// TIA Portal project "Quantum" (V16)

(* hardware
DEVICE "S7-1200 station_1"  S7-1200 Station
   slot 0: "Rack_0"  S7-1200 Rack  Rack  V1.0
   slot 1: "Quantum_Deshidratador"  CPU 1214C DC/DC/DC  6ES7 214-1AG40-0XB0  V4.4
   slot 101: "CM 1241 (RS422/485)_1"  6ES7 241-1CH32-0XB0  V2.1
*)

// ===== PLC "Quantum_Deshidratador"  CPU 1214C DC/DC/DC =====
// protected blocks, not shown: "MODULO_SECADOR"

VAR_GLOBAL   // PLC tag table "Default tag table"
   "Iniciar_Manual" AT %I0.0 : Bool;
   "Detener_Manual" AT %I0.1 : Bool;
   "Raw_Temperatura" AT %IW64 : Int;
   "Raw_Humedad" AT %IW66 : Int;
   "Deshidratador" AT %Q0.0 : Bool;
   "Actuador_Matte" AT %Q0.4 : Bool;
   "Ventiladores" AT %Q0.1 : Bool;
   "Resistencias" AT %Q0.5 : Bool;
   "Sensor_Modbus" AT %Q0.3 : Bool;
   "Sensor_HT" AT %Q0.2 : Bool;
   "System_Byte" AT %MB1 : Byte;
   "FirstScan" AT %M1.0 : Bool;
   "DiagStatusUpdate" AT %M1.1 : Bool;
   "AlwaysTRUE" AT %M1.2 : Bool;
   "AlwaysFALSE" AT %M1.3 : Bool;
   "Clock_Byte" AT %MB0 : Byte;
   "Clock_10Hz" AT %M0.0 : Bool;
   "Clock_5Hz" AT %M0.1 : Bool;
   "Clock_2.5Hz" AT %M0.2 : Bool;
   "Clock_2Hz" AT %M0.3 : Bool;
   "Clock_1.25Hz" AT %M0.4 : Bool;
   "Clock_1Hz" AT %M0.5 : Bool;
   "Clock_0.625Hz" AT %M0.6 : Bool;
   "Clock_0.5Hz" AT %M0.7 : Bool;
   "Control_Byte" AT %MB2 : Byte;
   "Detener" AT %M2.0 : Bool;
   "Iniciar" AT %M2.1 : Bool;
   "Pausar" AT %M2.2 : Bool;
   "Activar_Deshidratador" AT %M2.3 : Bool;
   "Limite_Matte" AT %M2.6 : Bool;
   "Sensor_Modbus_Manual" AT %M2.4 : Bool;
   "Set_Point_Deshidratador" AT %MD4 : Real;
   "Set_Point_Humedad" AT %MD8 : Real;
   "Iniciar_Pulse" AT %M40.0 : Bool;
   "Detener_Pulse" AT %M40.1 : Bool;
   "Guardar_Datos" AT %M40.2 : Bool;
   "Data_Log_Write_Error" AT %M40.3 : Bool;
   "Data_Log_Write_Busy" AT %M40.4 : Bool;
   "Data_Log_Write_Done" AT %M40.5 : Bool;
   "Data_Log_Write_Status" AT %MW96 : Word;
   "Clock_0.016Hz" AT %M40.6 : Bool;
   "Ret_Val" AT %MW98 : Int;
   "Sensor_HT_Manual" AT %M2.5 : Bool;
   "Actuador_Manual" AT %M2.7 : Bool;
   "Activar_Actuador" AT %M3.0 : Bool;
   "Tag_1" AT %M41.1 : Bool;
   "Habilitar_Matte" AT %M3.1 : Bool;
   "Set_Point_Limite" AT %MD12 : Real;
   "Humedad_Material_D11" AT %MD100 : Real;
   "Humedad_Material_D13" AT %MD104 : Real;
   "Humedad_Material_D16" AT %MD108 : Real;
   "Temp_D13" AT %MD114 : Real;
   "Temp_Matte" AT %MD118 : Real;
   "Hum_Matte" AT %MD62 : Real;
   "Temp_D11" AT %MD112 : Real;
   "Temp_Matte_Aux" AT %MD66 : Real;
   "Clock_Matte_Manual" AT %M41.2 : Bool;
   "Humedad_Material_D11_Ajuste" AT %MD70 : Real;
   "Humedad_Material_D13_Ajuste" AT %MD74 : Real;
   "Humedad_Material_D16_Ajuste" AT %MD78 : Real;
   "Hum_Matte_Aux" AT %MD82 : Real;
   "Random_Real_Seconds" AT %MD86 : Real;
   "Random_Status" AT %MW90 : Int;
   "Random_Sub_Status" AT %MW92 : Int;
   "Random_Error" AT %M3.2 : Bool;
   "Clock_Pulse" AT %M3.3 : Bool;
   "Randon_Dint_Seconds" AT %MD94 : DInt;
   "Tiempo_Histeresis_D1" AT %MD14 : Time;
   "Set_Point_Deshidratador1_Inicial" AT %MD18 : Real;
   "Set_Point_Deshidratador1_Intermedia" AT %MD22 : Real;
   "Set_Point_Deshidratador1_Final" AT %MD24 : Real;
   "Set_Point_Humedad_D1_Inicial" AT %MD28 : Real;
   "Set_Point_Humedad_D1_Intermedia" AT %MD32 : Real;
   "Set_Point_Humedad_D1_Final" AT %MD36 : Real;
   "Detener_Desde_Modo_Preset" AT %M41.3 : Bool;
   "Detener_Desde_Modo_Temporidado" AT %M41.4 : Bool;
END_VAR

VAR_GLOBAL CONSTANT   // PLC tag table "Default tag table"
   "Set_Point_Temp_Default" : Real := 55.0;
   "Set_Pont_Hum_Default" : Real := 5.0;
   "Set_Point_Lim_Default" : Real := -16.0;
   "Aux_Hum_D1" : Real := 10.0;
   "Aux_Hum_D4" : Real := 25.0;
   "Aux_Hum_D8" : Real := 25.0;
END_VAR

DATA_BLOCK "Modos_Operacion"   // DB32
{ S7_Optimized_Access := 'TRUE' }
VERSION : 0.1
   VAR RETAIN
      Modo_Preset_D1 : Bool := true;
      Momento_Actual_D1 : Int;
   END_VAR
BEGIN
END_DATA_BLOCK

DATA_BLOCK "Alarmas"   // DB44
{ S7_Optimized_Access := 'FALSE' }
VERSION : 0.1
   VAR
      Alarma_Fin_Operacion : Bool;
      Alarma_Fallo_Deh : Bool;
   END_VAR
BEGIN
END_DATA_BLOCK

// folder: Data Logging

DATA_BLOCK "CREAR_DB"   // DB7
{ S7_Optimized_Access := 'TRUE' }
VERSION : 0.1
   VAR
      records : UDInt := 17280;
      "name" : String := 'logging';
      id : DWord := 1;
      headers : String := 'HumD11,HumD13,HumD16,TempD11,TempD13,HumMatte,TempMatte';
      data : Struct
         humD11 : Real;
         humD13 : Real;
         humD16 : Real;
         tempD11 : Real;
         tempD13 : Real;
         humMatte : Real;
         tempMatte : Real;
      END_STRUCT;
      done : Bool;
      busy : Bool := true;
      error : Bool;
      status : Word;
   END_VAR
BEGIN
END_DATA_BLOCK

DATA_BLOCK "DATOS_VARIABLES"   // DB8
{ S7_Optimized_Access := 'FALSE' }
VERSION : 0.1
   VAR
      humD11 : Real;
      humD13 : Real;
      humD16 : Real;
      tempD11 : Real;
      tempD13 : Real;
      humMatte : Real;
      tempMatte : Real;
      dehRunning : Bool;
   END_VAR
BEGIN
END_DATA_BLOCK

DATA_BLOCK "Control_Log_DB"   // DB33
{ S7_Optimized_Access := 'FALSE' }
VERSION : 0.1
   VAR
      Iniciar_Log : Bool;
      Almacenar_Logs : Bool;
      Teminar_Log : Bool;
   END_VAR
BEGIN
END_DATA_BLOCK

// folder: Matte

DATA_BLOCK "DATOS_MODSEC"   // DB13
{ S7_Optimized_Access := 'TRUE' }
VERSION : 0.1
   VAR
      SimuHR : Int;
   END_VAR
   VAR RETAIN
      "Paso Control HR" : Time := T#5000ms;
      "Paso Grafica" : Time := T#10ms;
      "CRECIMIENTO HR" : Real := 80.0;
      TempMinHR : Real := 22.0;
   END_VAR
   VAR
      TempInf : Real := 0.0;
      TempSup : Real := 100.0;
      TempFilt : Real;
      TempFiltJP : Real;
      HRAux : Real;
      HRAuxJP : Real;
      HRFilt : Real;
      HRSim : Int;
      TempSim : Int;
      ProporcionHumedad : Real := 0.9;
      TempFiltCuar : Real;
      HRFiltCuar : Real;
      HRAuxCuar : Real;
   END_VAR
BEGIN
END_DATA_BLOCK

// folder: Modbus

DATA_BLOCK "MB_CONFIG"   // DB9
{ S7_Optimized_Access := 'FALSE' }
VERSION : 0.1
   VAR
      Again : Bool;
      Req : Bool;
      Mb_Addr : UInt := 1;
      Mode : USInt := 0;
      Data_Addr : UDInt := 40001;
      Data_Len : UInt := 5;
      Done : Bool;
      Busy : Bool;
      Error : Bool;
      Status : Word;
      Error_Status : Word;
      "Step" : Int := 1;
   END_VAR
BEGIN
END_DATA_BLOCK

DATA_BLOCK "MB_DATA_BUFFER"   // DB10
{ S7_Optimized_Access := 'FALSE' }
VERSION : 0.1
   VAR
      REGISTERS : Array[0..4] of UInt;
   END_VAR
BEGIN
END_DATA_BLOCK

DATA_BLOCK "MB_LOAD"   // DB11
{ S7_Optimized_Access := 'FALSE' }
VERSION : 0.1
   VAR
      Baud : UDInt := 9600;
      Parity : UDInt;
      Done : Bool;
      Error : Bool;
      Status : Word;
      Done_Stored : Bool;
      Error_Stored : Bool;
      Status_Error : Word;
   END_VAR
BEGIN
END_DATA_BLOCK

// folder: Sensores

DATA_BLOCK "Escalado_Temp_DB"   // DB18
{ S7_Optimized_Access := 'TRUE' }
VERSION : 0.1
// stored: InstanceOfName Escalado_Temp
"Escalado_Temp"
BEGIN
END_DATA_BLOCK

DATA_BLOCK "Conversor_4-20_0-20_DB"   // DB19
{ S7_Optimized_Access := 'TRUE' }
VERSION : 0.1
// stored: InstanceOfName Conversor_4-20_0-20
"Conversor_4-20_0-20"
BEGIN
END_DATA_BLOCK

DATA_BLOCK "Sensor_HR_DB"   // DB20
{ S7_Optimized_Access := 'TRUE' }
VERSION : 0.1
// stored: InstanceOfName Sensor_HR
"Sensor_HR"
BEGIN
END_DATA_BLOCK

DATA_BLOCK "Filtro_Promedio_DB"   // DB21
{ S7_Optimized_Access := 'TRUE' }
VERSION : 0.1
// stored: InstanceOfName Filtro_Promedio
"Filtro_Promedio"
BEGIN
END_DATA_BLOCK

DATA_BLOCK "Conversor_4-20_0-20_DB_1"   // DB22
{ S7_Optimized_Access := 'TRUE' }
VERSION : 0.1
// stored: InstanceOfName Conversor_4-20_0-20
"Conversor_4-20_0-20"
BEGIN
END_DATA_BLOCK

DATA_BLOCK "Simulacion_HR_DB"   // DB23
{ S7_Optimized_Access := 'TRUE' }
VERSION : 0.1
// stored: InstanceOfName Simulacion_HR
"Simulacion_HR"
BEGIN
END_DATA_BLOCK

DATA_BLOCK "Prom_FilterV2_DB"   // DB25
{ S7_Optimized_Access := 'TRUE' }
VERSION : 0.1
// stored: InstanceOfName Prom_FilterV2
"Prom_FilterV2"
BEGIN
END_DATA_BLOCK

DATA_BLOCK "Calibracion_Sensores"   // DB31
{ S7_Optimized_Access := 'TRUE' }
VERSION : 0.1
   VAR
      Ajuste_D11 : Real := 1.0;
      Ajuste_D13 : Real := 1.0;
      Ajuste_D16 : Real := 1.0;
      Ajuste_T1 : Real := 1.0;
   END_VAR
BEGIN
END_DATA_BLOCK

// folder: System blocks/Program resources

DATA_BLOCK "Paso_DB"   // DB1
{ S7_Optimized_Access := 'TRUE' }
AUTHOR : Simatic
FAMILY : IEC
NAME : IEC_TMR
VERSION : 1.0
// stored: InstanceOfName IEC_TIMER
"IEC_TIMER"
BEGIN
END_DATA_BLOCK

DATA_BLOCK "IEC_Timer_0_DB"   // DB14
{ S7_Optimized_Access := 'TRUE' }
AUTHOR : Simatic
FAMILY : IEC
NAME : IEC_TMR
VERSION : 1.0
// stored: InstanceOfName IEC_TIMER
"IEC_TIMER"
BEGIN
END_DATA_BLOCK

DATA_BLOCK "IEC_Timer_0_DB_1"   // DB16
{ S7_Optimized_Access := 'TRUE' }
AUTHOR : Simatic
FAMILY : IEC
NAME : IEC_TMR
VERSION : 1.0
// stored: InstanceOfName IEC_TIMER
"IEC_TIMER"
BEGIN
END_DATA_BLOCK

DATA_BLOCK "IEC_Timer_0_DB_2"   // DB17
{ S7_Optimized_Access := 'TRUE' }
AUTHOR : Simatic
FAMILY : IEC
NAME : IEC_TMR
VERSION : 1.0
// stored: InstanceOfName IEC_TIMER
"IEC_TIMER"
BEGIN
END_DATA_BLOCK

DATA_BLOCK "Timer_SimHR_DB"   // DB24
{ S7_Optimized_Access := 'TRUE' }
AUTHOR : Simatic
FAMILY : IEC
NAME : IEC_TMR
VERSION : 1.0
// stored: InstanceOfName IEC_TIMER
"IEC_TIMER"
BEGIN
END_DATA_BLOCK

DATA_BLOCK "IEC_Timer_0_DB_3"   // DB26
{ S7_Optimized_Access := 'TRUE' }
AUTHOR : Simatic
FAMILY : IEC
NAME : IEC_TMR
VERSION : 1.0
// stored: InstanceOfName IEC_TIMER
"IEC_TIMER"
BEGIN
END_DATA_BLOCK

DATA_BLOCK "Control_Temporizado"   // DB27
{ S7_Optimized_Access := 'TRUE' }
AUTHOR : Simatic
FAMILY : IEC
NAME : IEC_TMR
VERSION : 1.0
// stored: InstanceOfName IEC_TIMER
"IEC_TIMER"
BEGIN
END_DATA_BLOCK

DATA_BLOCK "IEC_Timer_0_DB_5"   // DB28
{ S7_Optimized_Access := 'TRUE' }
AUTHOR : Simatic
FAMILY : IEC
NAME : IEC_TMR
VERSION : 1.0
// stored: InstanceOfName IEC_TIMER
"IEC_TIMER"
BEGIN
END_DATA_BLOCK

DATA_BLOCK "IEC_Timer_0_DB_6"   // DB29
{ S7_Optimized_Access := 'TRUE' }
AUTHOR : Simatic
FAMILY : IEC
NAME : IEC_TMR
VERSION : 1.0
// stored: InstanceOfName IEC_TIMER
"IEC_TIMER"
BEGIN
END_DATA_BLOCK

DATA_BLOCK "IEC_Timer_0_DB_7"   // DB30
{ S7_Optimized_Access := 'TRUE' }
AUTHOR : Simatic
FAMILY : IEC
NAME : IEC_TMR
VERSION : 1.0
// stored: InstanceOfName IEC_TIMER
"IEC_TIMER"
BEGIN
END_DATA_BLOCK

DATA_BLOCK "Histeresis_Timer"   // DB34
{ S7_Optimized_Access := 'TRUE' }
AUTHOR : Simatic
FAMILY : IEC
NAME : IEC_TMR
VERSION : 1.0
// stored: InstanceOfName IEC_TIMER
"IEC_TIMER"
BEGIN
END_DATA_BLOCK

// folder: (top level)

FUNCTION "Control_Maestro" : Void   // FC1, SCL
{ S7_Optimized_Access := 'TRUE' }
VERSION : 0.1
   VAR_INPUT
      Temperatura : Int;
      SetValue : Int;
   END_VAR
   VAR_OUTPUT
      HabilitarControl : Bool;
      Resitencias : Bool;
   END_VAR
   VAR CONSTANT
      Hysteresis : Int := 1;
   END_VAR
BEGIN
   IF #Temperatura < #SetValue AND NOT #HabilitarControl OR #Temperatura > #SetValue + #Hysteresis AND #HabilitarControl THEN
       #HabilitarControl := FALSE;
       #Resitencias := TRUE;
   ELSE
       #HabilitarControl := TRUE;
       #Resitencias := FALSE;
   END_IF;
END_FUNCTION

ORGANIZATION_BLOCK "Main"   // OB1, LAD, ProgramCycle
TITLE = "Main Program Sweep (Cycle)"
{ S7_Optimized_Access := 'TRUE' }
VERSION : 0.1
   VAR_INPUT
      Initial_Call : Bool;   // Initial call of this OB
      Remanence : Bool;   // =True, if remanent data are available
   END_VAR
   VAR_TEMP   // added for the SCL form of the ladder/FBD networks
      _w1 : Bool;
      _w2 : Bool;
      _w3 : Bool;
   END_VAR
BEGIN

REGION Network 1: Iniciar Detener
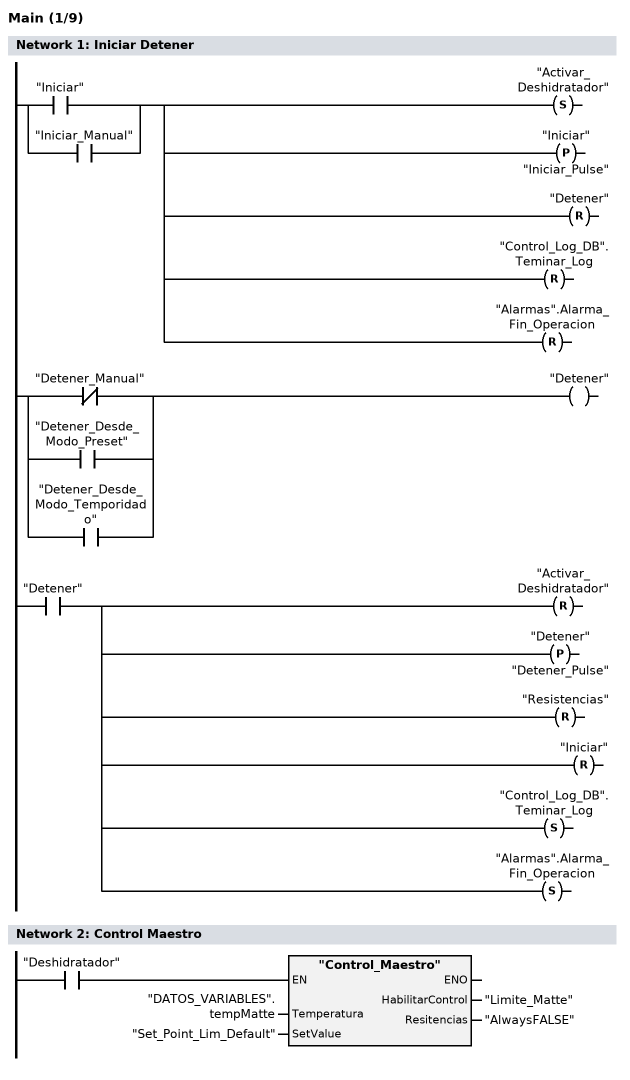
   #_w1 := "Iniciar" OR "Iniciar_Manual";
   IF #_w1 THEN "Activar_Deshidratador" := TRUE; END_IF;
   "Iniciar" := #_w1 AND NOT "Iniciar_Pulse";   // rising edge
   "Iniciar_Pulse" := #_w1;
   IF #_w1 THEN
       "Detener" := FALSE;
       "Control_Log_DB".Teminar_Log := FALSE;
       "Alarmas".Alarma_Fin_Operacion := FALSE;
   END_IF;
   "Detener" := NOT "Detener_Manual" OR "Detener_Desde_Modo_Preset" OR "Detener_Desde_Modo_Temporidado";
   IF "Detener" THEN "Activar_Deshidratador" := FALSE; END_IF;
   #_w2 := "Detener";
   #_w3 := "Detener";
   "Detener" := #_w2 AND NOT "Detener_Pulse";   // rising edge
   "Detener_Pulse" := #_w2;
   IF #_w3 THEN
       "Resistencias" := FALSE;
       "Iniciar" := FALSE;
       "Control_Log_DB".Teminar_Log := TRUE;
       "Alarmas".Alarma_Fin_Operacion := TRUE;
   END_IF;
END_REGION

REGION Network 2: Control Maestro
   RUNG wire#powerrail
      Contact( "Deshidratador" )
      "Control_Maestro"(Temperatura := "DATOS_VARIABLES".tempMatte, SetValue := "Set_Point_Lim_Default", HabilitarControl => "Limite_Matte", Resitencias => "AlwaysFALSE")
   END_RUNG
   // the same network as SCL:
   IF "Deshidratador" THEN
       "Control_Maestro"(Temperatura := "DATOS_VARIABLES".tempMatte,
                         SetValue := "Set_Point_Lim_Default",
                         HabilitarControl => "Limite_Matte",
                         Resitencias => "AlwaysFALSE");
   END_IF;
END_REGION

REGION Network 3: Matte
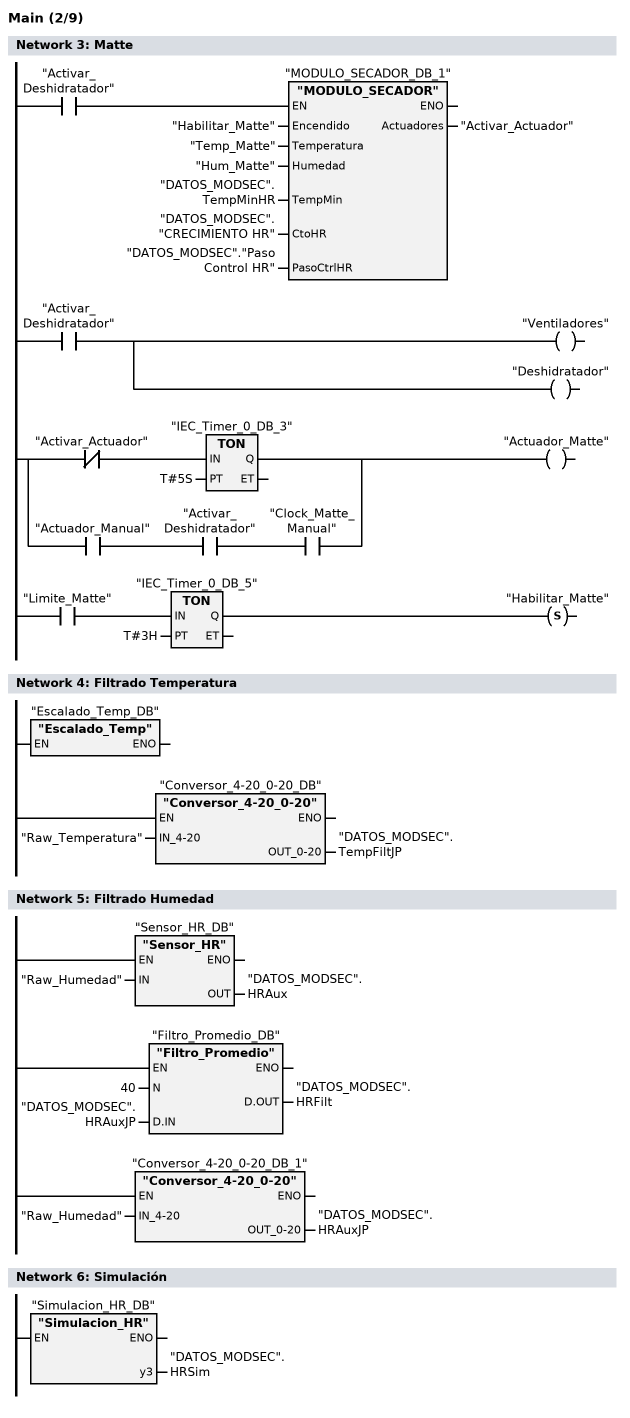
   IF "Activar_Deshidratador" THEN
       "MODULO_SECADOR_DB_1"(Encendido := "Habilitar_Matte",   // "MODULO_SECADOR"
                             Temperatura := "Temp_Matte",
                             Humedad := "Hum_Matte",
                             TempMin := "DATOS_MODSEC".TempMinHR,
                             CtoHR := "DATOS_MODSEC"."CRECIMIENTO HR",
                             PasoCtrlHR := "DATOS_MODSEC"."Paso Control HR",
                             Actuadores => "Activar_Actuador");
   END_IF;
   "Ventiladores" := "Activar_Deshidratador";
   "Deshidratador" := "Activar_Deshidratador";
   "IEC_Timer_0_DB_3".TON(IN := NOT "Activar_Actuador", PT := T#5S);
   "Actuador_Matte" := "IEC_Timer_0_DB_3".Q OR ("Actuador_Manual" AND "Activar_Deshidratador" AND "Clock_Matte_Manual");
   "IEC_Timer_0_DB_5".TON(IN := "Limite_Matte", PT := T#3H);
   IF "IEC_Timer_0_DB_5".Q THEN "Habilitar_Matte" := TRUE; END_IF;
END_REGION

REGION Network 4: Filtrado Temperatura
   RUNG wire#powerrail
      "Escalado_Temp_DB"()
   END_RUNG
   RUNG wire#powerrail
      "Conversor_4-20_0-20_DB"("IN_4-20" := "Raw_Temperatura", "OUT_0-20" => "DATOS_MODSEC".TempFiltJP)
   END_RUNG
   // the same network as SCL:
   "Escalado_Temp_DB"();   // "Escalado_Temp"
   "Conversor_4-20_0-20_DB"("IN_4-20" := "Raw_Temperatura", "OUT_0-20" => "DATOS_MODSEC".TempFiltJP);   // "Conversor_4-20_0-20"
END_REGION

REGION Network 5: Filtrado Humedad
   RUNG wire#powerrail
      "Sensor_HR_DB"(IN := "Raw_Humedad", OUT => "DATOS_MODSEC".HRAux)
   END_RUNG
   RUNG wire#powerrail
      "Filtro_Promedio_DB"(N := 40, "D.IN" := "DATOS_MODSEC".HRAuxJP, "D.OUT" => "DATOS_MODSEC".HRFilt)
   END_RUNG
   RUNG wire#powerrail
      "Conversor_4-20_0-20_DB_1"("IN_4-20" := "Raw_Humedad", "OUT_0-20" => "DATOS_MODSEC".HRAuxJP)
   END_RUNG
   // the same network as SCL:
   "Sensor_HR_DB"(IN := "Raw_Humedad", OUT => "DATOS_MODSEC".HRAux);   // "Sensor_HR"
   "Filtro_Promedio_DB"(N := 40, "D.IN" := "DATOS_MODSEC".HRAuxJP, "D.OUT" => "DATOS_MODSEC".HRFilt);   // "Filtro_Promedio"
   "Conversor_4-20_0-20_DB_1"("IN_4-20" := "Raw_Humedad", "OUT_0-20" => "DATOS_MODSEC".HRAuxJP);   // "Conversor_4-20_0-20"
END_REGION

REGION Network 6: Simulación
   RUNG wire#powerrail
      "Simulacion_HR_DB"(y3 => "DATOS_MODSEC".HRSim)
   END_RUNG
   // the same network as SCL:
   "Simulacion_HR_DB"(y3 => "DATOS_MODSEC".HRSim);   // "Simulacion_HR"
END_REGION

REGION Network 7: Manejo Sensorica
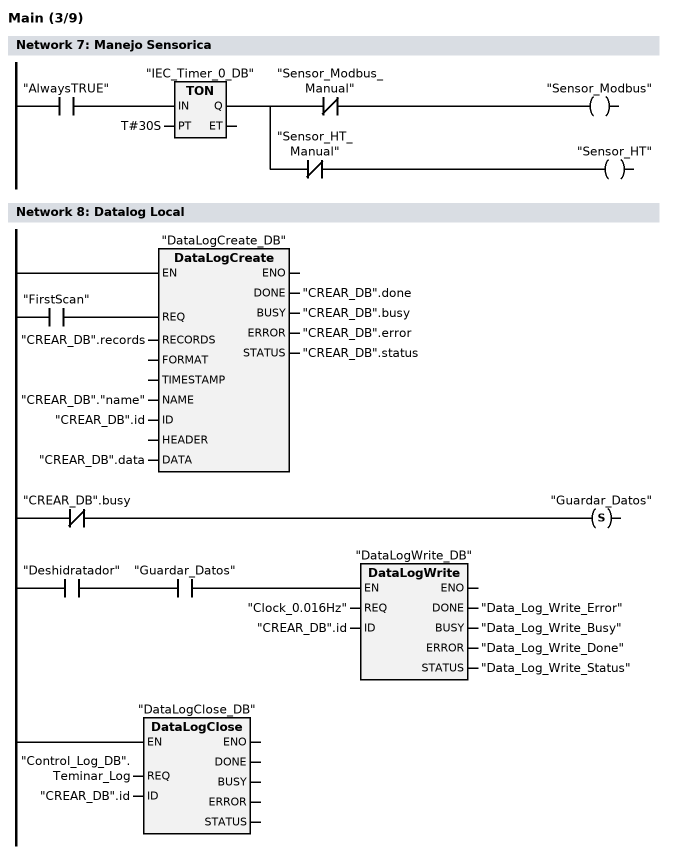
   "IEC_Timer_0_DB".TON(IN := "AlwaysTRUE", PT := T#30S);
   "Sensor_Modbus" := "IEC_Timer_0_DB".Q AND NOT "Sensor_Modbus_Manual";
   "Sensor_HT" := "IEC_Timer_0_DB".Q AND NOT "Sensor_HT_Manual";
END_REGION

REGION Network 8: Datalog Local
   "DataLogCreate_DB"(REQ := "FirstScan",   // DataLogCreate
                      RECORDS := "CREAR_DB".records,
                      "NAME" := "CREAR_DB"."name",
                      ID := "CREAR_DB".id,
                      DATA := "CREAR_DB".data,
                      DONE => "CREAR_DB".done,
                      BUSY => "CREAR_DB".busy,
                      ERROR => "CREAR_DB".error,
                      STATUS => "CREAR_DB".status);
   IF NOT "CREAR_DB".busy THEN "Guardar_Datos" := TRUE; END_IF;
   IF "Deshidratador" AND "Guardar_Datos" THEN
       "DataLogWrite_DB"(REQ := "Clock_0.016Hz",   // DataLogWrite
                         ID := "CREAR_DB".id,
                         DONE => "Data_Log_Write_Error",
                         BUSY => "Data_Log_Write_Busy",
                         ERROR => "Data_Log_Write_Done",
                         STATUS => "Data_Log_Write_Status");
   END_IF;
   "DataLogClose_DB"(REQ := "Control_Log_DB".Teminar_Log, ID := "CREAR_DB".id);   // DataLogClose
END_REGION

REGION Network 9: Mover Datos para Log Remoto
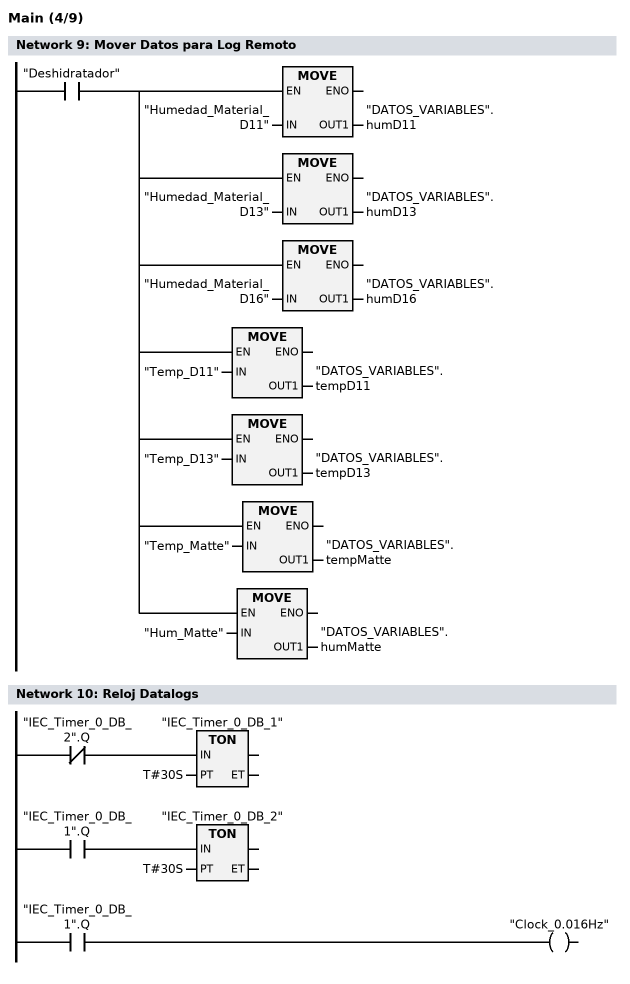
   RUNG wire#powerrail
      Contact( "Deshidratador" )
      wire#w1
      Move(in := "Humedad_Material_D11", out1 => "DATOS_VARIABLES".humD11)
   END_RUNG
   RUNG wire#w1
      Move(in := "Humedad_Material_D13", out1 => "DATOS_VARIABLES".humD13)
   END_RUNG
   RUNG wire#w1
      Move(in := "Humedad_Material_D16", out1 => "DATOS_VARIABLES".humD16)
   END_RUNG
   RUNG wire#w1
      Move(in := "Temp_D11", out1 => "DATOS_VARIABLES".tempD11)
   END_RUNG
   RUNG wire#w1
      Move(in := "Temp_D13", out1 => "DATOS_VARIABLES".tempD13)
   END_RUNG
   RUNG wire#w1
      Move(in := "Temp_Matte", out1 => "DATOS_VARIABLES".tempMatte)
   END_RUNG
   RUNG wire#w1
      Move(in := "Hum_Matte", out1 => "DATOS_VARIABLES".humMatte)
   END_RUNG
   // the same network as SCL:
   IF "Deshidratador" THEN
       "DATOS_VARIABLES".humD11 := "Humedad_Material_D11";
       "DATOS_VARIABLES".humD13 := "Humedad_Material_D13";
       "DATOS_VARIABLES".humD16 := "Humedad_Material_D16";
       "DATOS_VARIABLES".tempD11 := "Temp_D11";
       "DATOS_VARIABLES".tempD13 := "Temp_D13";
       "DATOS_VARIABLES".tempMatte := "Temp_Matte";
       "DATOS_VARIABLES".humMatte := "Hum_Matte";
   END_IF;
END_REGION

REGION Network 10: Reloj Datalogs
   "IEC_Timer_0_DB_1".TON(IN := NOT "IEC_Timer_0_DB_2".Q, PT := T#30S);
   "IEC_Timer_0_DB_2".TON(IN := "IEC_Timer_0_DB_1".Q, PT := T#30S);
   "Clock_0.016Hz" := "IEC_Timer_0_DB_1".Q;
END_REGION

REGION Network 11: Mover Datos para Log Local
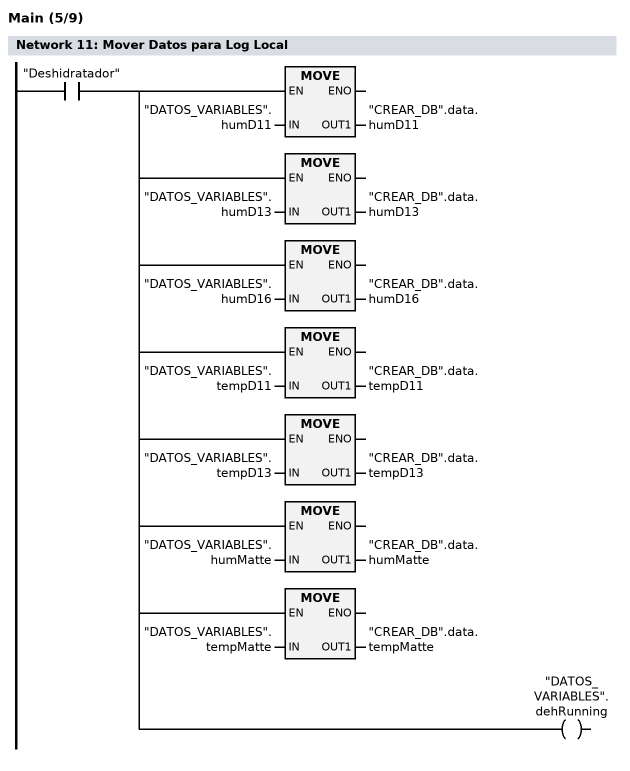
   RUNG wire#powerrail
      Contact( "Deshidratador" )
      wire#w1
      Move(in := "DATOS_VARIABLES".humD11, out1 => "CREAR_DB".data.humD11)
   END_RUNG
   RUNG wire#w1
      Move(in := "DATOS_VARIABLES".humD13, out1 => "CREAR_DB".data.humD13)
   END_RUNG
   RUNG wire#w1
      Move(in := "DATOS_VARIABLES".humD16, out1 => "CREAR_DB".data.humD16)
   END_RUNG
   RUNG wire#w1
      Move(in := "DATOS_VARIABLES".tempD11, out1 => "CREAR_DB".data.tempD11)
   END_RUNG
   RUNG wire#w1
      Move(in := "DATOS_VARIABLES".tempD13, out1 => "CREAR_DB".data.tempD13)
   END_RUNG
   RUNG wire#w1
      Move(in := "DATOS_VARIABLES".humMatte, out1 => "CREAR_DB".data.humMatte)
   END_RUNG
   RUNG wire#w1
      Move(in := "DATOS_VARIABLES".tempMatte, out1 => "CREAR_DB".data.tempMatte)
   END_RUNG
   RUNG wire#w1
      Coil( "DATOS_VARIABLES".dehRunning )
   END_RUNG
   // the same network as SCL:
   IF "Deshidratador" THEN
       "CREAR_DB".data.humD11 := "DATOS_VARIABLES".humD11;
       "CREAR_DB".data.humD13 := "DATOS_VARIABLES".humD13;
       "CREAR_DB".data.humD16 := "DATOS_VARIABLES".humD16;
       "CREAR_DB".data.tempD11 := "DATOS_VARIABLES".tempD11;
       "CREAR_DB".data.tempD13 := "DATOS_VARIABLES".tempD13;
       "CREAR_DB".data.humMatte := "DATOS_VARIABLES".humMatte;
       "CREAR_DB".data.tempMatte := "DATOS_VARIABLES".tempMatte;
   END_IF;
   "DATOS_VARIABLES".dehRunning := "Deshidratador";
END_REGION

REGION Network 12: Comunicación Modbus
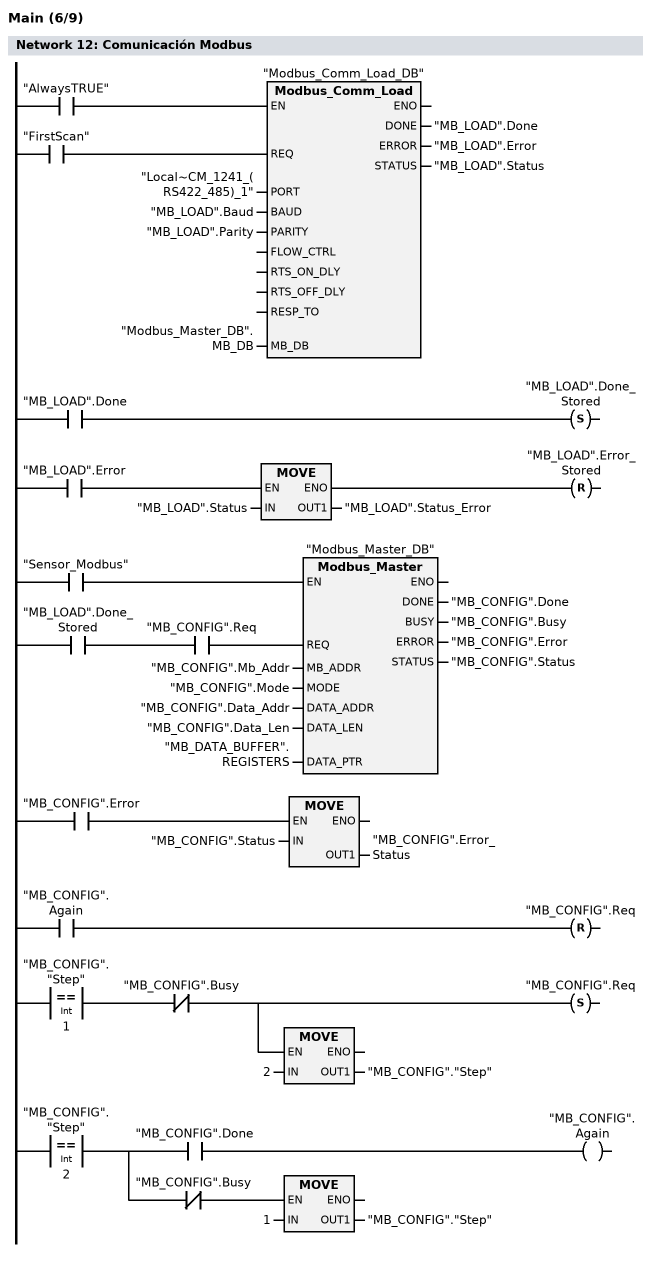
   IF "AlwaysTRUE" THEN
       "Modbus_Comm_Load_DB"(REQ := "FirstScan",   // Modbus_Comm_Load
                             PORT := "Local~CM_1241_(RS422_485)_1",
                             BAUD := "MB_LOAD".Baud,
                             PARITY := "MB_LOAD".Parity,
                             MB_DB := "Modbus_Master_DB".MB_DB,
                             DONE => "MB_LOAD".Done,
                             ERROR => "MB_LOAD".Error,
                             STATUS => "MB_LOAD".Status);
   END_IF;
   IF "MB_LOAD".Done THEN "MB_LOAD".Done_Stored := TRUE; END_IF;
   IF "MB_LOAD".Error THEN
       "MB_LOAD".Status_Error := "MB_LOAD".Status;
       "MB_LOAD".Error_Stored := FALSE;
   END_IF;
   IF "Sensor_Modbus" THEN
       "Modbus_Master_DB"(REQ := "MB_LOAD".Done_Stored AND "MB_CONFIG".Req,   // Modbus_Master
                          MB_ADDR := "MB_CONFIG".Mb_Addr,
                          MODE := "MB_CONFIG".Mode,
                          DATA_ADDR := "MB_CONFIG".Data_Addr,
                          DATA_LEN := "MB_CONFIG".Data_Len,
                          DATA_PTR := "MB_DATA_BUFFER".REGISTERS,
                          DONE => "MB_CONFIG".Done,
                          BUSY => "MB_CONFIG".Busy,
                          ERROR => "MB_CONFIG".Error,
                          STATUS => "MB_CONFIG".Status);
   END_IF;
   IF "MB_CONFIG".Error THEN "MB_CONFIG".Error_Status := "MB_CONFIG".Status; END_IF;
   IF "MB_CONFIG".Again THEN "MB_CONFIG".Req := FALSE; END_IF;
   IF ("MB_CONFIG"."Step" = 1) AND NOT "MB_CONFIG".Busy THEN
       "MB_CONFIG".Req := TRUE;
       "MB_CONFIG"."Step" := 2;
   END_IF;
   #_w1 := "MB_CONFIG"."Step" = 2;
   "MB_CONFIG".Again := #_w1 AND "MB_CONFIG".Done;
   IF #_w1 AND NOT "MB_CONFIG".Busy THEN "MB_CONFIG"."Step" := 1; END_IF;
END_REGION

REGION Network 13: Escalización Humedad
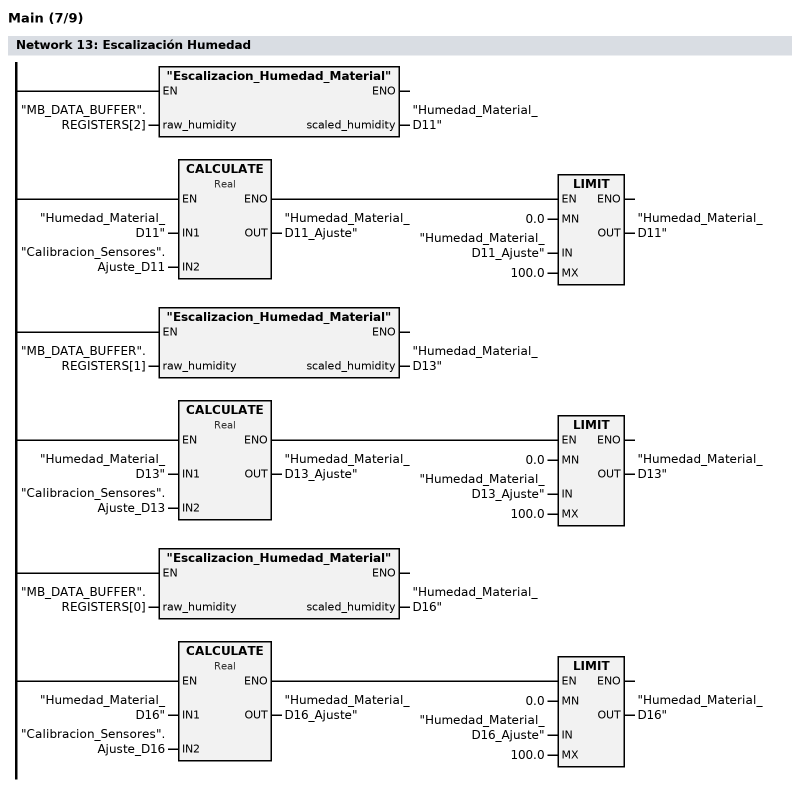
   "Escalizacion_Humedad_Material"(raw_humidity := "MB_DATA_BUFFER".REGISTERS[2],
                           scaled_humidity => "Humedad_Material_D11");
   "Humedad_Material_D11_Ajuste" := "Humedad_Material_D11" - "Calibracion_Sensores".Ajuste_D11;
   "Humedad_Material_D11" := LIMIT(MN := 0.0, IN := "Humedad_Material_D11_Ajuste", MX := 100.0);
   "Escalizacion_Humedad_Material"(raw_humidity := "MB_DATA_BUFFER".REGISTERS[1],
                           scaled_humidity => "Humedad_Material_D13");
   "Humedad_Material_D13_Ajuste" := "Humedad_Material_D13" - "Calibracion_Sensores".Ajuste_D13;
   "Humedad_Material_D13" := LIMIT(MN := 0.0, IN := "Humedad_Material_D13_Ajuste", MX := 100.0);
   "Escalizacion_Humedad_Material"(raw_humidity := "MB_DATA_BUFFER".REGISTERS[0],
                           scaled_humidity => "Humedad_Material_D16");
   "Humedad_Material_D16_Ajuste" := "Humedad_Material_D16" - "Calibracion_Sensores".Ajuste_D16;
   "Humedad_Material_D16" := LIMIT(MN := 0.0, IN := "Humedad_Material_D16_Ajuste", MX := 100.0);
END_REGION

REGION Network 14: Humedad y Temperatura Deshidratador
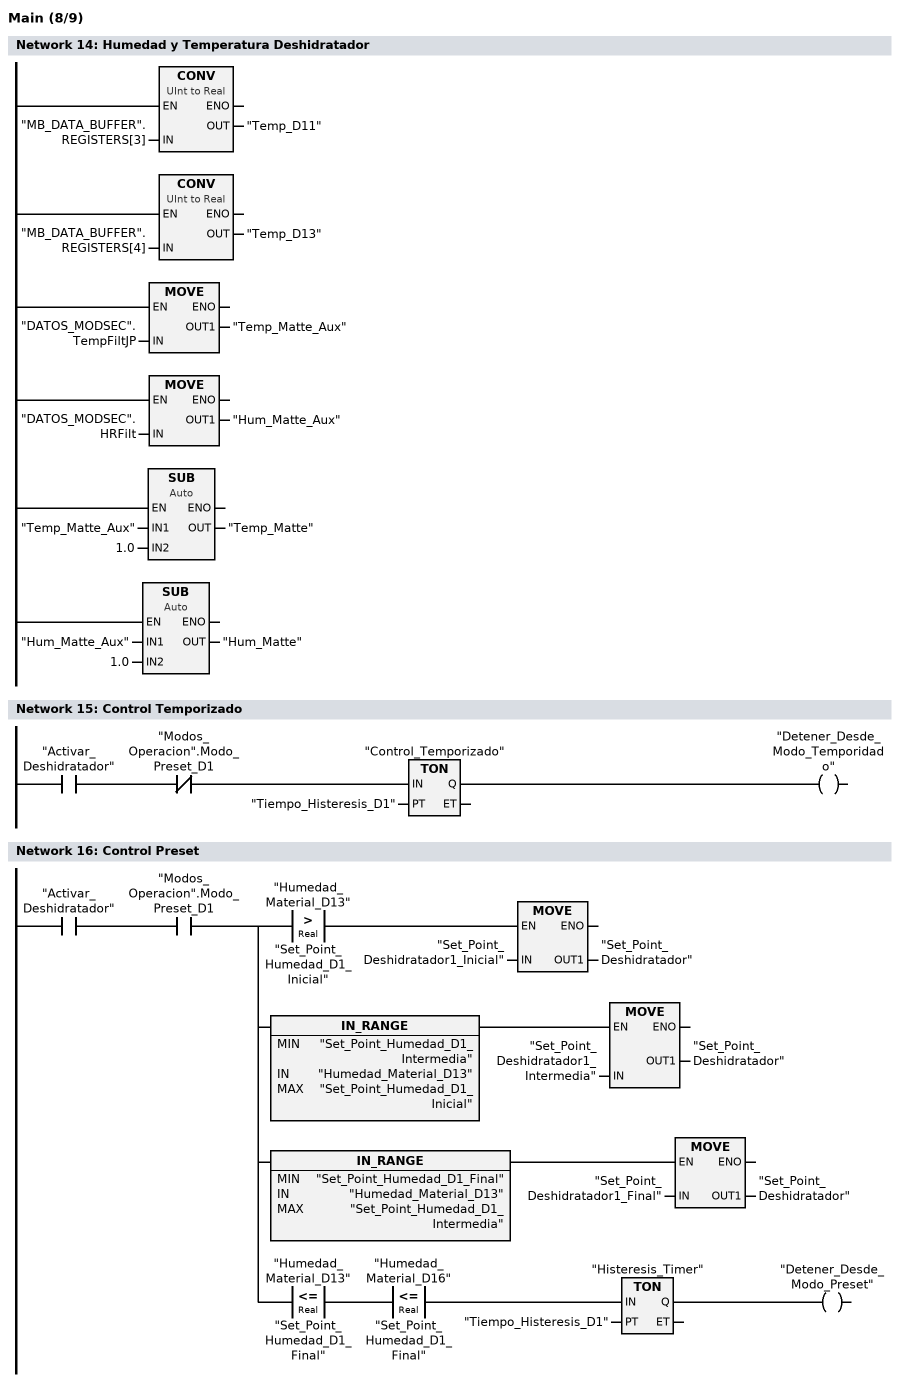
   RUNG wire#powerrail
      { S7_Templates := "[SrcType := UInt, DestType := Real]" } Convert(in := "MB_DATA_BUFFER".REGISTERS[3], out => "Temp_D11")
   END_RUNG
   RUNG wire#powerrail
      { S7_Templates := "[SrcType := UInt, DestType := Real]" } Convert(in := "MB_DATA_BUFFER".REGISTERS[4], out => "Temp_D13")
   END_RUNG
   RUNG wire#powerrail
      Move(in := "DATOS_MODSEC".TempFiltJP, out1 => "Temp_Matte_Aux")
   END_RUNG
   RUNG wire#powerrail
      Move(in := "DATOS_MODSEC".HRFilt, out1 => "Hum_Matte_Aux")
   END_RUNG
   RUNG wire#powerrail
      Sub(in1 := "Temp_Matte_Aux", in2 := 1.0, out => "Temp_Matte")
   END_RUNG
   RUNG wire#powerrail
      Sub(in1 := "Hum_Matte_Aux", in2 := 1.0, out => "Hum_Matte")
   END_RUNG
   // the same network as SCL:
   "Temp_D11" := UINT_TO_REAL("MB_DATA_BUFFER".REGISTERS[3]);
   "Temp_D13" := UINT_TO_REAL("MB_DATA_BUFFER".REGISTERS[4]);
   "Temp_Matte_Aux" := "DATOS_MODSEC".TempFiltJP;
   "Hum_Matte_Aux" := "DATOS_MODSEC".HRFilt;
   "Temp_Matte" := "Temp_Matte_Aux" - 1.0;
   "Hum_Matte" := "Hum_Matte_Aux" - 1.0;
END_REGION

REGION Network 15: Control Temporizado
   "Control_Temporizado".TON(IN := "Activar_Deshidratador" AND NOT "Modos_Operacion".Modo_Preset_D1,
                           PT := "Tiempo_Histeresis_D1");
   "Detener_Desde_Modo_Temporidado" := "Control_Temporizado".Q;
END_REGION

REGION Network 16: Control Preset
   #_w1 := "Activar_Deshidratador" AND "Modos_Operacion".Modo_Preset_D1;
   IF #_w1 AND ("Humedad_Material_D13" > "Set_Point_Humedad_D1_Inicial") THEN
       "Set_Point_Deshidratador" := "Set_Point_Deshidratador1_Inicial";
   END_IF;
   IF #_w1 AND ("Set_Point_Humedad_D1_Intermedia" <= "Humedad_Material_D13") AND ("Humedad_Material_D13" <= "Set_Point_Humedad_D1_Inicial") THEN
       "Set_Point_Deshidratador" := "Set_Point_Deshidratador1_Intermedia";
   END_IF;
   IF #_w1 AND ("Set_Point_Humedad_D1_Final" <= "Humedad_Material_D13") AND ("Humedad_Material_D13" <= "Set_Point_Humedad_D1_Intermedia") THEN
       "Set_Point_Deshidratador" := "Set_Point_Deshidratador1_Final";
   END_IF;
   "Histeresis_Timer".TON(IN := #_w1 AND ("Humedad_Material_D13" <= "Set_Point_Humedad_D1_Final") AND ("Humedad_Material_D16" <= "Set_Point_Humedad_D1_Final"),
                          PT := "Tiempo_Histeresis_D1");
   "Detener_Desde_Modo_Preset" := "Histeresis_Timer".Q;
END_REGION

REGION Network 17: Carga Pagina Definida por Usuario
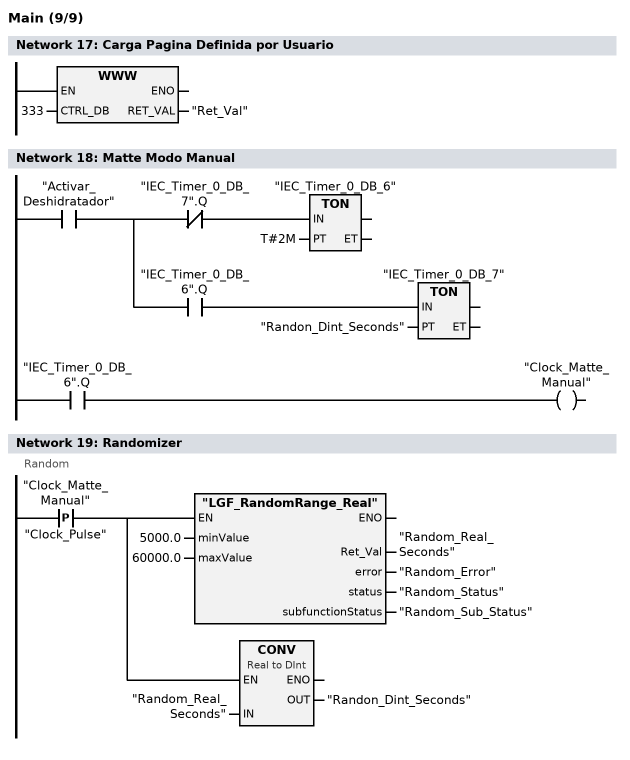
   "Ret_Val" := WWW(CTRL_DB := 333);
END_REGION

REGION Network 18: Matte Modo Manual
   "IEC_Timer_0_DB_6".TON(IN := "Activar_Deshidratador" AND NOT "IEC_Timer_0_DB_7".Q, PT := T#2M);
   "IEC_Timer_0_DB_7".TON(IN := "Activar_Deshidratador" AND "IEC_Timer_0_DB_6".Q, PT := "Randon_Dint_Seconds");
   "Clock_Matte_Manual" := "IEC_Timer_0_DB_6".Q;
END_REGION

REGION Network 19: Randomizer
   // Random
   RUNG wire#powerrail
      P_Contact(operand := "Clock_Matte_Manual", bit := "Clock_Pulse")
      wire#w1
      "LGF_RandomRange_Real"(minValue := 5000.0, maxValue := 60000.0, Ret_Val => "Random_Real_Seconds", error => "Random_Error", status => "Random_Status", subfunctionStatus => "Random_Sub_Status")
   END_RUNG
   RUNG wire#w1
      { S7_Templates := "[SrcType := Real, DestType := DInt]" } Convert(in := "Random_Real_Seconds", out => "Randon_Dint_Seconds")
   END_RUNG
   // the same network as SCL:
   #_w1 := "Clock_Matte_Manual" AND NOT "Clock_Pulse";   // rising edge of "Clock_Matte_Manual"
   "Clock_Pulse" := "Clock_Matte_Manual";
   IF #_w1 THEN
       "Random_Real_Seconds" := "LGF_RandomRange_Real"(minValue := 5000.0,
                               maxValue := 60000.0,
                               error => "Random_Error",
                               status => "Random_Status",
                               subfunctionStatus => "Random_Sub_Status");
       "Randon_Dint_Seconds" := REAL_TO_DINT("Random_Real_Seconds");
   END_IF;
END_REGION
END_ORGANIZATION_BLOCK

ORGANIZATION_BLOCK "Cyclic interrupt"   // OB30, LAD, CyclicInterrupt
{ S7_Optimized_Access := 'TRUE' }
VERSION : 0.1
   VAR_INPUT
      Initial_Call : Bool;   // Initial call of this OB
      Event_Count : Int;   // Events discarded
   END_VAR
BEGIN

REGION Network 1
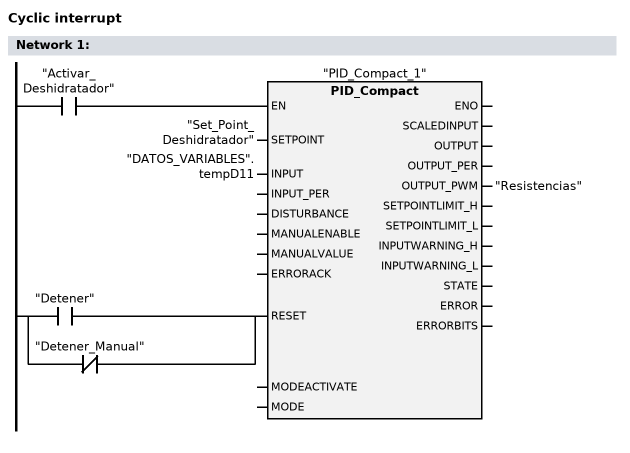
   IF "Activar_Deshidratador" THEN
       "PID_Compact_1"(Setpoint := "Set_Point_Deshidratador",   // PID_Compact
                       Input := "DATOS_VARIABLES".tempD11,
                       Reset := "Detener" OR NOT "Detener_Manual",
                       Output_PWM => "Resistencias");
   END_IF;
END_REGION
END_ORGANIZATION_BLOCK

// folder: LGF/4 Math operations

FUNCTION "LGF_RandomRange_Real" : Real   // FC10014, SCL
TITLE = LGF_RandomRange_Real
{ S7_Optimized_Access := 'TRUE' }
AUTHOR : Siemens_Digital_Industries
FAMILY : LGF
NAME : LGF_RandomRange_Real
// This function generates a random value in defined limits with each call.  
// The random number has the data type Real in the specified range.
// Diese Funktion generiert bei jedem Aufruf einen zufälligen Wert zwischen einem definierten Max- und Minwert.  
// Die Zufallszahl hat den Datentyp Real im spezifiziertem Wertebereich.
   VAR_INPUT
      minValue : Real;   // Minimalwert der für den Wertebereich der Zufallszahl - Untergrenze / Minimum value of the range of the random number - lower border
      maxValue : Real;   // Maximalwert der für den Wertebereich der Zufallszahl - Obergrenze / Maximum value of the range of the random number - upper border
   END_VAR
   VAR_OUTPUT
      error : Bool;   // FALSE: No error TRUE: An error occurred during the execution of the FB / FALSE: Kein Fehler TRUE: Während der Ausführung des FB ist ein Fehler aufgetreten
      status : Word;   // 16#0000-16#7FFF: Status of the FB 16#8000-16#FFFF: Error identification (see following Table) / 16#0000-16#7FFF: Status des FB 16#8000-16#FFFF: Fehleridentifikation (siehe folgende Tabelle)
      subfunctionStatus : Word;   // Status or return value of called FB's, FC's and system blocks / Status oder Rückgabewert von aufgerufenen FB's / FC's und Systemfunktionen
   END_VAR
   VAR_TEMP
      tempTime : DTL;   // Temp memory for System time / Temp variable für System Zeit
      tempNanoSecondInDWord : DWord;   // Temp UDInt converted to DWord for access to individual bytes / Temp UDInt konvertiert nach Dword für den Zufriff per Slice auf die Bytes
      tempTimeStatus : Word;   // Temp status of the instruction `RD_SYS_T` / Temp Status der Systemfunktion `RD_SYS_T`
      tempRandomValue : DWord;   // Temp Random startvalue / Temp Zufallswert als Startwert
      tempNormReal : Real;   // Temp normalized Real value (0.0 - 1.0) / Temp Normalisierer Realwert (0.0 - 1.0)
   END_VAR
   // Ret_Val : Random Real number in the predefined range / Zufallszahl vom Datentyp Real im definierten Wertebereich
   VAR CONSTANT
      ZERO : Real := 0.0;   // Zero / 0.0 - value in case of error / Null / 0.0 - Rückgabewert im Fehlerfall
      MAX_UDINT : UDInt := 4294967295;   // Maximum UDInt datatype / Maximalwert eines UDInt Datentype
      SUB_STATUS_NO_ERROR : Word := 16#0000;   // Status: sub function call ends without error / Status: Unterfunktionsaufruf ohne Fehler beendet
      STATUS_FINISHED_NO_ERROR : Word := 16#0000;   // Execution finished without errors / Abarbeitung ohne Fehler beendet
      ERR_MAX_LESS_MIN : Word := 16#8200;   // Error: The ranges specified are wrong: `minValue` is greater than `maxValue` / Fehler: Der spezifizierte Wetebereich is fehlerhaft: `minValue` ist größer als `maxValue`
      ERR_RD_SYS_T : Word := 16#8600;   // Error in `RD_SYS_T` command - check `subFunctionStatus` code / Fehler in Anweisung `RD_SYS_T` - weitere infos in `subFunctionStatus`
   END_VAR
BEGIN
   REGION Block info header
     //=============================================================================
     // SIEMENS AG / (c)Copyright 2017
     //-----------------------------------------------------------------------------
     // Title:            LGF_RandomRange_Real
     // Comment/Function: This function generates random numbers in defined limits (Datatype Real)
     // Library/Family:   LGF(Library General Functions)
     // Author:           Siemens Digital Industry Support
     // Tested with:      S7-PLCSIM Advanced V2.0 SP1
     // Engineering:      TIA Portal V15 Update 2
     // Restrictions:     ENO disabled - error handling done by error and status
     // Requirements:     PLC (S7-1200 / S7-1500)
     //-------------------------------------------------------------------------------
     // Change log table:
     // Version  | Date       | Expert in charge       | Changes applied
     //----------|------------|------------------------|------------------------------
     // 01.00.00 19.08.2015  Siemens Industry Online Support
     //                      First released version
     // 01.00.01 02.01.2017  Siemens Industry Online Support
     //                      Upgrade: TIA Portal V14 Update 1
     // 01.00.02 02.03.2017  Siemens Industry Online Support
     //                      Bugfix: FC number
     // 01.00.03 17.08.2018  Siemens Industry Online Support
     //                      Upgrade: TIA V15 Update 2
     // 01.00.04 23.11.2018  Siemens Industry Online Support
     //                      Upgrade: TIA V15.1
     // 01.01.00 13.11.2019  Simatic Systems Support
     //                      Renamed from "LGF_RandomReal" to "LGF_RandomRange_Real"
     //                      Regions, comments and constants are added
     // 03.00.00 23.04.2020  Simatic Systems Support
     //                      Set version to V3.0.0, harmonize the version of the whole library
     // 03.00.01 04.02.2021  Simatic Systems Support
     //                      Insert documentation
     //=============================================================================
   END_REGION Block info header

   REGION DESCRIPTION
     (/*Note
   :    The status of called commands is output in `subFunctionStatus`. In this case, the output value in `status` indicates which command caused the error. In this case, refer to the TIA Portal Online Help section for information on the respective commands.

   The block generates random values that are between the specified `minValue` and the `maxValue`. This random value is output via the `Ret_Val`.

   The random value is formed from the nanoseconds of the current system time of the CPU. The byte order of this value is inverted and then converted to a floating point.
   Hinweis
   :    In `subFunctionStatus` wird der Status von aufgerufenen Anweisungen ausgegeben. Der Ausgangswert in `status` gibt in diesem Fall an, welche Anweisung den Fehler verursacht hat. Holen Sie sich in diesem Fall die Informationen aus der TIA Portal Online Hilfe zu den jeweiligen Anweisungen.

   Der Baustein generiert zufällige Werte, die zwischen dem angegebenen `minValue`-Wert und `maxValue`-Wert liegen. Dieser zufällige Wert wird über den `Ret_Val` ausgegeben.

   Der Zufallswert wird aus den Nanosekunden der aktuellen Systemzeit der CPU gebildet. Dabei wird die Bytereihenfolge dieses Wertes invertiert und anschließend in eine Gleitkommazahl ungewandelt.*/)
   END_REGION DESCRIPTION

   REGION Validation
     // Check if the maximal Value is less than the minimal value
     IF (#minValue > #maxValue) THEN
       #error := true;
       #status := #ERR_MAX_LESS_MIN;
       #subfunctionStatus := #SUB_STATUS_NO_ERROR;
       #LGF_RandomRange_Real := #ZERO;
       RETURN;
     END_IF;

     // Read system time
     #tempTimeStatus := INT_TO_WORD(RD_SYS_T(#tempTime));

     // Check return variable for error
     IF (#tempTimeStatus <> #SUB_STATUS_NO_ERROR) THEN
       #error := true;
       #status := #ERR_RD_SYS_T;
       #subfunctionStatus := #tempTimeStatus;
       #LGF_RandomRange_Real := #ZERO;
       RETURN;
     END_IF;
   END_REGION

   REGION Calculating random number
     // Converting to double word so individual bytes can be addressed
     #tempNanoSecondInDWord := UDINT_TO_DWORD(#tempTime.NANOSECOND);

     // Calculate a random-start-value depending on the time
     #tempRandomValue.%B3 := #tempNanoSecondInDWord.%B0;
     #tempRandomValue.%B2 := #tempNanoSecondInDWord.%B1;
     #tempRandomValue.%B1 := #tempNanoSecondInDWord.%B2;
     #tempRandomValue.%B0 := #tempNanoSecondInDWord.%B3;

     // Norm the calculated random number: 0.0 <= #tempNormReal <= 1.0
     #tempNormReal := UDINT_TO_REAL(DWORD_TO_UDINT(#tempRandomValue)) / UDINT_TO_REAL(#MAX_UDINT);

     // Scale the tempNormReal to be in the range of maxValue and minValue
     #LGF_RandomRange_Real := ((#tempNormReal * (#maxValue - #minValue) + (#minValue)));

     #error := false;
     #status := #STATUS_FINISHED_NO_ERROR;
     #subfunctionStatus := #SUB_STATUS_NO_ERROR;
     // ENO mechanism is not used
     ENO := TRUE;
   END_REGION
END_FUNCTION

// folder: Sensores

FUNCTION_BLOCK "Escalado_Temp"   // FB2, SCL
{ S7_Optimized_Access := 'TRUE' }
VERSION : 0.1
   VAR
      TempAux : Real;
   END_VAR
   VAR CONSTANT
      M_Time : Time := T#20ms;
   END_VAR
BEGIN
   #TempAux := INT_TO_REAL("Raw_Temperatura");
   //#TempAux := INT_TO_REAL("DATOS_MODSEC".TempSim);

   "Prom_FilterV2_DB"(Scale_Value:=#TempAux,
                      Inf_Limit:="DATOS_MODSEC".TempInf,
                      Sup_Limit:="DATOS_MODSEC".TempSup,
                      Filter_Set_Time:=#M_Time,
                      Max_Analog_Value:=27648,
                      Prom_Filter=>"DATOS_MODSEC".TempFilt);
END_FUNCTION_BLOCK

FUNCTION_BLOCK "Conversor_4-20_0-20"   // FB3, SCL
{ S7_Optimized_Access := 'TRUE' }
VERSION : 0.1
   VAR_INPUT
      "IN_4-20" : Word;
   END_VAR
   VAR_OUTPUT
      "OUT_0-20" : Real;
   END_VAR
BEGIN
   #"OUT_0-20" := (#"IN_4-20" / 221.0) - 25.0;
END_FUNCTION_BLOCK

FUNCTION_BLOCK "Sensor_HR"   // FB27, SCL
{ S7_Optimized_Access := 'TRUE' }
VERSION : 0.1
   VAR_INPUT
      IN : Int;
   END_VAR
   VAR_OUTPUT
      OUT : Real;
   END_VAR
BEGIN
   // Normalización y Escalado Sensor 4-20mA
   #OUT := SCALE_X(MIN := 0.0,
                   VALUE := NORM_X(MIN := 0,
                                   VALUE := #IN,   // <--- Entrada Sensor Valor Int
                                   MAX := 27648),
                   MAX := 100.0);
END_FUNCTION_BLOCK

FUNCTION_BLOCK "Filtro_Promedio"   // FB28, SCL
{ S7_Optimized_Access := 'TRUE' }
VERSION : 0.1
   VAR_INPUT
      N : Int;
      "D.IN" : Real;
   END_VAR
   VAR_OUTPUT
      "D.OUT" : Real;
   END_VAR
   VAR
      D : Array[0..100] of Real;
      I : Int;
      J : Int;
      "D.Sum" : Real;
   END_VAR
BEGIN
   // Procesamiento de Valor Promedio 
   // Tiempo de cilco 100ms <- From Cyclic interrupt [OB30]
   // #N = 60  <- 60*100ms = 6 segundos  (10*0.1s = 1Seg)

   // --- Almacenamiento de los Datos -----
   #I :=(#I + 1) MOD #N;   // <- 0 .. N = N+1 Datos
   #D[#I] := #"D.IN";      // NOTA: La posición #D[N] nunca se utiliza

   // --- Calculo del valor Promedio --------------------------------------
   #"D.Sum" := 0;
   FOR #J := 0 TO (#N-1) BY 1 DO
       #"D.Sum" := #"D.Sum" + #D[#J];
   END_FOR;

   #"D.OUT" := #"D.Sum" / #N;
END_FUNCTION_BLOCK

FUNCTION_BLOCK "Simulacion_HR"   // FB29, SCL
{ S7_Optimized_Access := 'TRUE' }
VERSION : 0.1
   VAR_OUTPUT
      y3 : Int;
   END_VAR
   VAR
      Timer_SimHR : Struct
         IN : Bool;
         PT : Time;
         Q : Bool;
         ET : Time;
      END_STRUCT;
      t : Int;
      t2 : Real;
      y3_Aux : Int;
   END_VAR
BEGIN
   IF #Timer_SimHR.IN = FALSE
   THEN
       #Timer_SimHR.IN := TRUE;
   END_IF;
   IF #Timer_SimHR.Q = TRUE AND #Timer_SimHR.IN = TRUE
   THEN
       #Timer_SimHR.IN := FALSE;
       #t := (#t + 1) MOD 3160;
       #t2 := INT_TO_REAL(#t);
       #t2 := #t2 / 100;
       //#y1_Aux := REAL_TO_INT((1000 * (SIN(#t2))) + 10000);  // Temperatura Superior
       //#y2_Aux := REAL_TO_INT((1000 * (SIN(#t2 + 10))) + 40 + 10000);    // Temperatura Inferior
       #y3_Aux := REAL_TO_INT((1000 * (SIN(#t2 + 20))) + 40 + 10 + 20000);   // Humedad Relativa
       #y3 := #y3_Aux;
   END_IF;

   "Timer_SimHR_DB".TON(IN:=#Timer_SimHR.IN,
                        PT:="DATOS_MODSEC"."Paso Grafica",
                        Q=>#Timer_SimHR.Q,
                        ET=>#Timer_SimHR.ET);
END_FUNCTION_BLOCK

FUNCTION_BLOCK "Prom_FilterV2"   // FB40, SCL
{ S7_Optimized_Access := 'TRUE' }
VERSION : 0.1
   VAR_INPUT
      Scale_Value : Real;
      Inf_Limit : Real;
      Sup_Limit : Real;
      Cal : Real;
      Filter_Set_Time : Time;
      Max_Analog_Value : UInt;
   END_VAR
   VAR_OUTPUT
      Prom_Filter : Real;
   END_VAR
   VAR
      i : Int;
   END_VAR
   VAR RETAIN
      i_Acum : Real;
   END_VAR
   VAR
      Pv_Value : Real;
      Pv_Aux1 : Real;
      En_Filter_Timer : Bool := False;
      Filter_P_Time : Time;
      Filter_TImer : TONR_TIME;
   END_VAR
BEGIN
   #Filter_TImer(IN:=NOT(#En_Filter_Timer),
                 R:=#En_Filter_Timer,
                 PT:=#Filter_Set_Time,
                 Q=>#En_Filter_Timer,
                 ET=>#Filter_P_Time);

   // "Filter_Timer".TONR(IN:=NOT(#En_Filter_Timer),
   //                     R:=#En_Filter_Timer,
   //                     PT:=#Filter_Set_Time,
   //                     Q=>#En_Filter_Timer,
   //                     ET=>#Filter_P_Time);

   IF #En_Filter_Timer = True
   THEN
       IF #Scale_Value > 27648
       THEN
           #Prom_Filter := -1;
       ELSE
           FOR #i := 1 TO 200 DO
               #Pv_Aux1 := (NORM_X_REAL(MIN:=0, VALUE:= REAL_TO_INT(#Scale_Value), MAX:= #Max_Analog_Value));
               #Pv_Value := ((SCALE_X_REAL(MIN:=#Inf_Limit, VALUE:= #Pv_Aux1, MAX:= #Sup_Limit)) - #Cal);
               #i_Acum:= #i_Acum + #Pv_Value;
           END_FOR;
       END_IF;
       #i:=#i+1;
       #En_Filter_Timer := False;
   END_IF;

   IF #i >= 200
   THEN
       #Prom_Filter := #i_Acum / 200;
       #i_Acum := 0;
       #i:= 0;
   END_IF;
END_FUNCTION_BLOCK

FUNCTION "Escalizacion_Humedad_Material" : Void   // FC2, SCL
{ S7_Optimized_Access := 'TRUE' }
VERSION : 0.1
   VAR_INPUT
      raw_humidity : UInt;
   END_VAR
   VAR_OUTPUT
      scaled_humidity : UInt;
   END_VAR
   VAR_TEMP
      slope : Real;
   END_VAR
   VAR CONSTANT
      max_output : Real := 100.0;
      min_output : Real := 0.0;
      max_input : Real := 0.0;
      min_input : Real := 1023.0;
   END_VAR
BEGIN
   #slope := (#max_output - #min_output) / (#max_input - #min_input);
   #scaled_humidity := #slope * (UINT_TO_REAL(#raw_humidity) - #min_input) + #min_output;
END_FUNCTION